PROGRAM MAIN
VAR
	fbSlicer : FB_Slicer;
	bStartButton : BOOL;
	fM1Position : LREAL;
	fM1sPosition : LREAL;
	fM2Position : LREAL;
	nErrorID : UDINT;
END_VAR

fbSlicer(bStartButton := bStartButton,
		 fM1Position => fM1Position,
		 fM1sPosition => fM1sPosition,
		 fM2Position => fM2Position,
		 nErrorID => nErrorID);

END_PROGRAM

(* stored: Version 1.1.0.1, ProductVersion 3.1.4024.12
   POU MAIN: Id {487d2b30-aca7-4d70-bcc8-562be4c283ec}, SpecialFunc None *)
